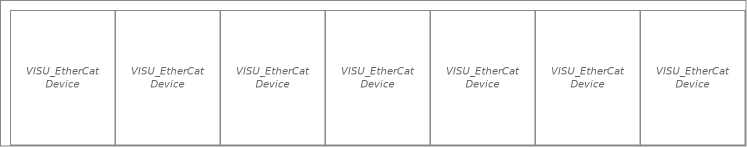
VISUALIZATION VISU_SafetyDomeAccessIO  // 747x147
VAR_IN_OUT
	ref : SafetyDomeAccessIO;
    widget : SafetyDomeAccessIOWidget;
END_VAR
    Frame (10,10 105x135)
        shows VISU_EtherCatDevice(device := ref.parts.COU, widget := widget.COU)
    Frame (115,10 105x135)
        shows VISU_EtherCatDevice(device := ref.parts.DI1, widget := widget.DI1)
    Frame (220,10 105x135)
        shows VISU_EtherCatDevice(device := ref.parts.DI2, widget := widget.DI2)
    Frame (325,10 105x135)
        shows VISU_EtherCatDevice(device := ref.parts.DO1, widget := widget.DO1)
    Frame (535,10 105x135)
        shows VISU_EtherCatDevice(device := ref.parts.RE1, widget := widget.RE1)
    Frame (640,10 105x135)
        shows VISU_EtherCatDevice(device := ref.parts.RE2, widget := widget.RE2)
    Frame (430,10 105x135)
        shows VISU_EtherCatDevice(device := ref.parts.SI1, widget := widget.SI1)
END_VISUALIZATION

(* stored: Version 1.1.0.1, ProductVersion 3.1.4019.2
   Visu VISU_SafetyDomeAccessIO: Id {ff47bd85-0ed6-4df1-b1ee-1ecd5cc26ce1} *)
